RoboDK station: Custom_Assistive_UR5e.rdk

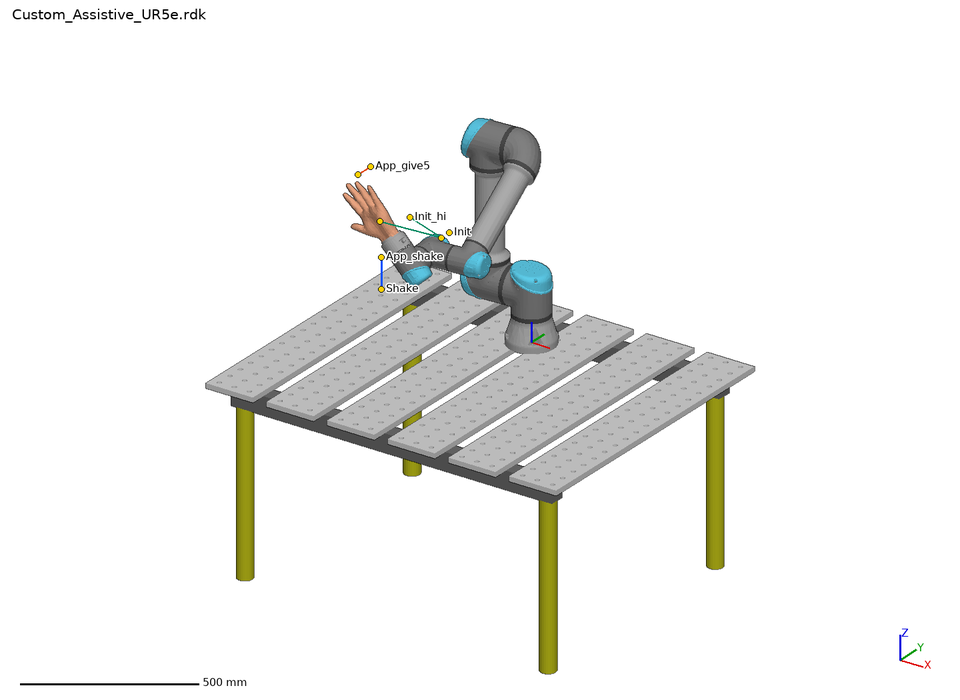
[picture v0: the station drawn from its stored meshes, robots at their saved joint values, targets as dots, program paths as lines]
Station Assistive_UR5e_SW (saved by RoboDK 5.9.2). Poses are relative to the parent item; angles as X-Y-Z fixed-axis rotations.
  - frame UR5e Base at (0, 0, 0) mm
    - robot UR5e: 6 axes, payload 5 kg, reach 850 mm, repeatability 0.03 mm, weight 18.4 kg
        modified DH rows (alpha deg, a mm, theta deg, d mm): 0, 0, 0, 162.5; 90, 0, 180, 0; 0, 425, 0, 0; 0, 392.25, 0, 133.3; -90, 0, 0, 99.7; 90, 0, 180, 99.6
        joint limits [-360, -360, -360, -360, -360, -360] to [360, 360, 360, 360, 360, 360]; home [0, -90, -90, 0, 90, 0]; saved at [-86.2, -89.19, -122.01, 301.2, -48.17, 76.05]
      - tool Hand, TCP at (0, 0, 50) mm, size 54.8 x 155.9 x 193.5 mm, geometry from Hand.stl
  - frame World at (0, 0, 0) mm
    - object Table at (0, 0, 0) mm, size 1193.8 x 965.2 x 609.6 mm, geometry from welding_table.sld
    - target Init (Cartesian target) at (0, -400, 500) mm, rotated rx 90 ry 0 rz 0 deg; joints [-57.836, -65.392, -107.167, 172.559, -57.836, 0] of UR5e
    - target App_shake (joint target) at (-300, -300, 300) mm, rotated rx 90 ry 0 rz 0 deg; joints [-129.97, -84.968, -123.366, -151.667, -129.97, 0] of UR5e
    - target Shake (joint target) at (-300, -300, 200) mm, rotated rx 90 ry 0 rz 0 deg; joints [-129.97, -95.332, -131.473, -133.195, -129.97, 0] of UR5e
    - target App_give5 (joint target) at (-380.86, -238.62, 533.82) mm, rotated rx 0 ry 0 rz 90 deg; joints [-130.679, -89.195, -122.013, 301.208, -90, 130.679] of UR5e
    - target Give5 (joint target) at (-380.86, -300, 533.82) mm, rotated rx 0 ry 0 rz 90 deg; joints [-125.814, -94.091, -116.939, 301.03, -90, 125.814] of UR5e
    - target Init_hi (Cartesian target) at (-107.87, -437.32, 533.82) mm, rotated rx -1.23 ry -0.31 rz 79.86 deg; joints [-86.2, -89.19, -122.01, 301.2, -88.73, 76.06] of UR5e
    - target Hi_right (Cartesian target) at (-5.01, -430.49, 495.73) mm, rotated rx 40.98 ry 9.25 rz 83.31 deg; joints [-86.2, -89.19, -122.01, 301.2, -131.83, 76.05] of UR5e
    - target Hi_left (Cartesian target) at (-204.11, -443.71, 495.73) mm, rotated rx -40.98 ry -9.25 rz 83.31 deg; joints [-86.2, -89.19, -122.01, 301.2, -48.17, 76.05] of UR5e
  - program Init (3 instructions, listed below)
  - program Hand_shake (5 instructions, listed below)
  - program Give_me_5! (5 instructions, listed below)
  - program MainProgram (4 instructions, listed below)
  - program Hi (7 instructions, listed below)
  - Python program Custom_Assistive_SW (listed below)
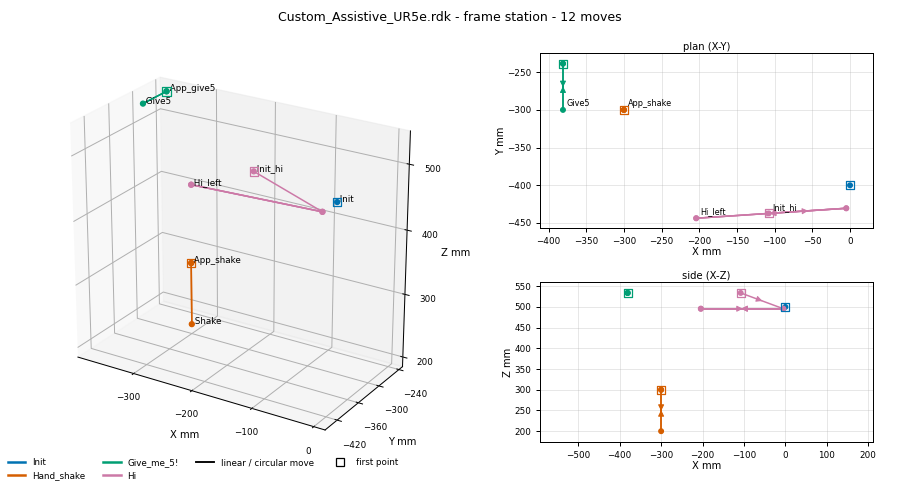
[picture p0: tool path of Custom_Assistive_UR5e.rdk in frame station, 12 of 12 moves have a stored position in this frame; points joined in program order, loops and branches not executed]

--- program Init (robot UR5e) ---
  Est. Ref.: UR5e Base
  Est. herr: Hand
  MoveJ (Init)

--- program Hand_shake (robot UR5e) ---
  Est. Ref.: UR5e Base
  Est. herr: Hand
  MoveL (App_shake)
  MoveL (Shake)
  MoveL (App_shake)

--- program Give_me_5! (robot UR5e) ---
  Est. Ref.: UR5e Base
  Est. herr: Hand
  MoveL (App_give5)
  MoveL (Give5)
  MoveL (App_give5)

--- program MainProgram (robot UR5e) ---
  Llamar Init
  Llamar Hand_shake
  Llamar Give_me_5!
  Llamar Init

--- program Hi (robot UR5e) ---
  Set Ref.: UR5e Base
  Set Tool: Hand
  MoveJ (Init_hi)
  MoveL (Hi_right)
  MoveL (Hi_left)
  MoveL (Hi_right)
  MoveL (Hi_left)

--- Python program Custom_Assistive_SW ---
import os
import time
import tkinter as tk
from tkinter import messagebox
from robodk.robolink import *
from robodk.robomath import *

# Define relative path to the .rdk file
relative_path = "src/roboDK/Assistive_UR5e.rdk"
absolute_path = os.path.abspath(relative_path)

# Start RoboDK with the project file
RDK = Robolink()
RDK.AddFile(absolute_path)

# Retrieve items from the RoboDK station
robot = RDK.Item("UR5e")
base = RDK.Item("UR5e Base")
tool = RDK.Item("Hand")
Init_target = RDK.Item("Init")
App_shake_target = RDK.Item("App_shake")
Shake_target = RDK.Item("Shake")
App_give5_target = RDK.Item("App_give5")
Give5_target = RDK.Item("Give5")
Init_hi_target = RDK.Item("Init_hi")
Hi_left_target = RDK.Item("Hi_left")
Hi_right_target = RDK.Item("Hi_right")

# Set robot frame, tool and speed
robot.setPoseFrame(base)
robot.setPoseTool(tool)
robot.setSpeed(20)

# Move to initial position
def move_to_init():
    print("Init")
    robot.MoveL(Init_target, True)
    print("Init_target REACHED")

# Perform handshake sequence
def hand_shake():
    print("Hand Shake")
    robot.MoveL(App_shake_target, True)
    robot.MoveL(Shake_target, True)
    robot.MoveL(App_shake_target, True)
    print("Hand Shake FINISHED")

# Perform "Give me 5" sequence
def give_me_5():
    print("Give me 5!")
    robot.MoveL(App_give5_target, True)
    robot.MoveL(Give5_target, True)
    robot.MoveL(App_give5_target, True)
    print("Give me 5! FINISHED")

# Perform "Hi" sequence
def say_hi():
    print("Saying Hi!")
    robot.MoveL(Init_hi_target, True)
    robot.MoveL(Hi_right_target, True)
    robot.MoveL(Hi_left_target, True)
    robot.MoveL(Hi_right_target, True)
    robot.MoveL(Hi_left_target, True)
    print("Saying Hi! FINISHED")

# Main sequence
def main():
    say_hi()

# Confirmation dialog to close RoboDK
def confirm_close():
    root = tk.Tk()
    root.withdraw()
    response = messagebox.askquestion(
        "Close RoboDK",
        "Do you want to save changes before closing RoboDK?",
        icon='question'
    )
    if response == 'yes':
        RDK.Save()
        RDK.CloseRoboDK()
        print("RoboDK saved and closed.")
    else:
        RDK.CloseRoboDK()
        print("RoboDK closed without saving.")

# Run main and handle closing
if __name__ == "__main__":
    main()
    #confirm_close()
